// TIA Portal V15.1 export
// export: Created 2020-06-12T07:35:47.4443359Z, ExportSetting None, DisplayName Totally Integrated Automation Portal, DisplayVersion V15.1, DisplayName TIA Portal Openness, DisplayVersion V15.1, DisplayName STEP 7 Professional, DisplayVersion V15.1, DisplayName STEP 7 Safety, DisplayVersion V15.1, DisplayName WinCC Advanced, DisplayVersion V15.1
FUNCTION "GAS_zaux" : Void   // FC51, FBD
{ S7_Optimized_Access := 'TRUE' }
// stored: SetENOAutomatically False
BEGIN

REGION Network 1: EV08: Gas for Alloy addition
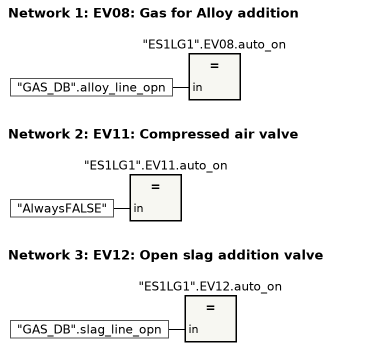
   "ES1LG1".EV08.auto_on := "GAS_DB".alloy_line_opn;
END_REGION

REGION Network 2: EV11: Compressed air valve
   // This valve has no function in this project. Always open
   "ES1LG1".EV11.auto_on := "AlwaysFALSE";
END_REGION

REGION Network 3: EV12: Open slag addition valve
   "ES1LG1".EV12.auto_on := "GAS_DB".slag_line_opn;
END_REGION
END_FUNCTION
